Universal Robots PolyScope program: L03_Touchoff.urp

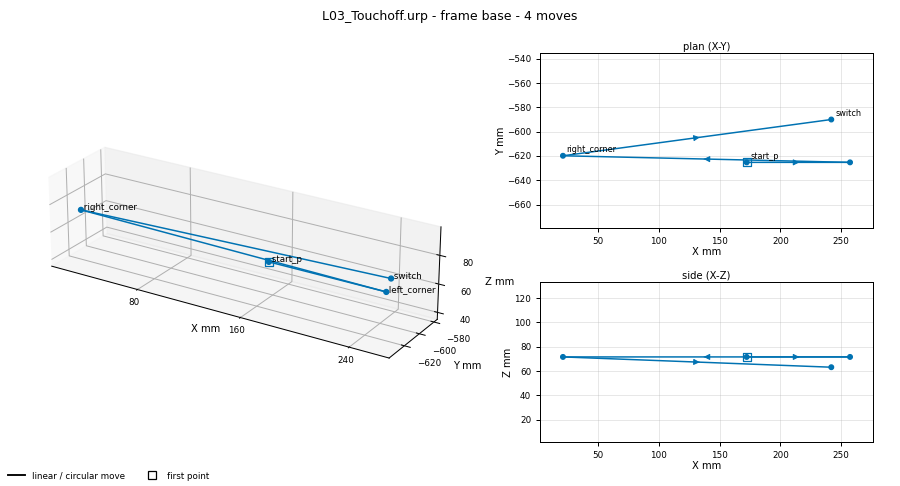
[picture p0: tool path of L03_Touchoff.urp in frame base, 4 of 6 moves have a stored position in this frame; points joined in program order, loops and branches not executed]
Program L03_Touchoff (installation=default directory=/programs createdIn=5.9.1.1031110 lastSavedIn=5.9.1.1031110 robotSerialNumber=20195501059)
Calibrated DH parameters: a=[0.000146, -0.418764, -0.053981, 0.000058, -0.000023, 0]; d=[0.162545, 37.319448, -206.067439, 168.881546, 0.09955, 0.099464]; alpha=[1.57004, -0.001979, 0.002304, 1.570607, -1.57066, 0]; deltaTheta=[0, -0.174616, -1.258233, 1.432844, -0.000001, 0]
BeforeStart
  init_p := get_actual_tcp_pose()
  MoveL speed 250 mm/s, acceleration 1200 mm/s^2 (useActiveTCP=true) feature=Base
    Waypoint Waypoint (Variable): variable=init_p
  If init_p[2]<0.100
    safe_p := p[init_p[0],init_p[1],0.100,init_p[3],init_p[4],init_p[5]]
    MoveL speed 250 mm/s, acceleration 1200 mm/s^2 (useActiveTCP=true) feature=Base
      Waypoint Waypoint (Variable): variable=safe_p
Robot Program (runOnlyOnce=true)
  MoveJ speed 60 deg/s, acceleration 80 deg/s^2 (useActiveTCP=true) feature=Base
    Waypoint start_p: TCP in base x=172.194 y=-625.301 z=71.57 mm, rx=2.2093 ry=2.2334 rz=0 rad; joints [93.486, -62.74, 92.599, -119.853, 270.005, 92.879] deg; TCP offset x=0 y=0 z=174 mm, rx=0 ry=0 rz=0 rad
    URCap Gripper (Robotiq_Grippers, Robotiq Inc.) dataModel(position=100.0, force=5.0, speed=30.0, positionInDouble=100.0, forceInDouble=5.0, speedInDouble=30.0, slaveIds=[9], blocking=true)
  MoveL speed 250 mm/s, acceleration 1200 mm/s^2 (useActiveTCP=true) feature=Base
    Waypoint left_corner: TCP in base x=257.245 y=-625.305 z=71.59 mm, rx=2.2093 ry=2.2334 rz=-0.0001 rad; joints [100.944, -59.419, 87.293, -117.871, 269.995, 100.334] deg
    MoveDirectionNode (selectedDirection=ZMinus toolParams=0.01, 0.8)
      Until TOOL_CONTACT_DETECTION (allowActions=true retraction=0)
        left_z := get_actual_tcp_pose()
    MoveDirectionNode (selectedDirection=ZPlus)
      Until DISTANCE (allowActions=false deceleration=3 distanceNodeType=STOP) Distance=0.02; motionParameters(blendRadius=0)
    Waypoint right_corner: TCP in base x=21.033 y=-619.88 z=71.59 mm, rx=2.2093 ry=2.2334 rz=-0.0001 rad; joints [79.481, -66.113, 97.801, -121.684, 270.016, 78.878] deg
    MoveDirectionNode (selectedDirection=ZMinus toolParams=0.01, 0.8)
      Until TOOL_CONTACT_DETECTION (allowActions=true retraction=0)
        right_z := get_actual_tcp_pose()
    MoveDirectionNode (selectedDirection=ZPlus)
      Until DISTANCE (allowActions=false deceleration=3 distanceNodeType=STOP) Distance=0.02; motionParameters(blendRadius=0)
    Waypoint switch: TCP in base x=241.822 y=-590.044 z=63.127 mm, rx=2.2094 ry=2.2334 rz=0.0001 rad; joints [100.168, -63.448, 95.144, -121.687, 270.011, 99.567] deg
    MoveDirectionNode (selectedDirection=ZMinus toolParams=0.01, 0.8)
      Until TOOL_CONTACT_DETECTION (allowActions=true retraction=0)
        switch_z := get_actual_tcp_pose()
    MoveDirectionNode (selectedDirection=ZPlus)
      Until DISTANCE (allowActions=false deceleration=3 distanceNodeType=STOP) Distance=0.02; motionParameters(blendRadius=0)
